INTERFACE I_Nodes

METHOD PUBLIC Accept
VAR_INPUT
	Visitor : I_NodeVisitor;
END_VAR
END_METHOD

PROPERTY PUBLIC Count : DINT
GET
END_GET
END_PROPERTY

METHOD PUBLIC GetById : I_Node
VAR_INPUT
	Id : NodeId;
END_VAR
END_METHOD

METHOD PUBLIC GetByIndex : I_Node
VAR_INPUT
	Id : NodeId;
END_VAR
END_METHOD

METHOD PUBLIC GetFirst : I_Node
END_METHOD

METHOD PUBLIC GetHighestExecutionOrder : DINT
VAR_INPUT
END_VAR
END_METHOD

METHOD PUBLIC GetNext : I_Node
VAR_INPUT
	CurrentNode : I_Node;
END_VAR
END_METHOD

END_INTERFACE

(* stored: Version 1.1.0.1, ProductVersion 3.1.4024.12
   Itf I_Nodes: Id {b3c6ceaf-e729-05e3-0d25-7dba72f18e8c}
   Method Accept: Id {6416c07f-9d21-07ac-09c2-e94e2357b99e}
   Property Count: Id {20c4e3cd-c93e-00c6-085e-148464fff949}
   Get Get: Id {2eb952aa-241a-03cf-1874-34592f8cb09c}
   Method GetById: Id {40137c31-a513-0265-3cd0-61225f7b79b7}
   Method GetByIndex: Id {abc22edb-160c-06b4-3513-ffd84ef8ec35}
   Method GetFirst: Id {feddbc3f-4e18-0f11-38ed-c4eba56c857b}
   Method GetHighestExecutionOrder: Id {edfdd55f-8e55-0283-19f7-6fc1afffb08c}
   Method GetNext: Id {1b2591ca-aae4-0122-37f3-8d91f1aa64cb} *)
